// Mitsubishi GX Works2 project: 21   PLC: FX3G

// task Task_01 (event TRUE, interval 0, priority 31): POU_01

PROGRAM POU_01
VAR
  gas : INT;
  ton1 : TON;
END_VAR
IF M8002 THEN
	gas := 0;
END_IF;

	IF M0=TRUE THEN
	gas:=11;
END_IF;

IF M1=TRUE THEN
	gas:=21;
END_IF;

IF M2=TRUE THEN
	gas:=31;
END_IF;

CASE gas OF

	11:
	Y0:=TRUE;
	Y1:=FALSE;
	Y2:=FALSE;
	Y3:=FALSE;
	ton1(IN := NOT ton1.Q, PT := T#0.5s);
	IF ton1.Q THEN
		gas:=12;
	END_IF;
	
	12:
	Y0:=FALSE;
	Y1:=TRUE;
	Y2:=FALSE;
	Y3:=FALSE;
	ton1(IN := NOT ton1.Q, PT := T#0.5s);
	IF ton1.Q THEN
		gas:=13;
	END_IF;

 13:
	Y0:=FALSE;
	Y1:=FALSE;
	Y2:=TRUE;
	Y3:=FALSE;
	ton1(IN := NOT ton1.Q, PT := T#0.5s);
	IF ton1.Q THEN
		gas:=14;
	END_IF;
	
	14:
	Y0:=FALSE;
	Y1:=FALSE;
	Y2:=FALSE;
	Y3:=TRUE;
	ton1(IN := NOT ton1.Q, PT := T#0.5s);
	IF ton1.Q THEN
		gas:=11;
	END_IF;
	
	21:
	Y0:=TRUE;
	Y1:=FALSE;
	Y2:=FALSE;
	Y3:=FALSE;
	ton1(IN := NOT ton1.Q, PT := T#1s);
	IF ton1.Q THEN
		gas:=22;
	END_IF;
	
	22:
	Y0:=FALSE;
	Y1:=TRUE;
	Y2:=FALSE;
	Y3:=FALSE;
	ton1(IN := NOT ton1.Q, PT := T#1s);
	IF ton1.Q THEN
		gas:=23;
	END_IF;

 	23:
	Y0:=FALSE;
	Y1:=FALSE;
	Y2:=TRUE;
	Y3:=FALSE;
	ton1(IN := NOT ton1.Q, PT := T#1s);
	IF ton1.Q THEN
		gas:=24;
	END_IF;
	
	24:
	Y0:=FALSE;
	Y1:=FALSE;
	Y2:=FALSE;
	Y3:=TRUE;
	ton1(IN := NOT ton1.Q, PT := T#1s);
	IF ton1.Q THEN
		gas:=21;
	END_IF;
	
	31:
	Y0:=TRUE;
	Y1:=FALSE;
	Y2:=FALSE;
	Y3:=FALSE;
	ton1(IN := NOT ton1.Q, PT := T#1.5s);
	IF ton1.Q THEN
		gas:=32;
	END_IF;
	
	32:
	Y0:=FALSE;
	Y1:=TRUE;
	Y2:=FALSE;
	Y3:=FALSE;
	ton1(IN := NOT ton1.Q, PT := T#1.5s);
	IF ton1.Q THEN
		gas:=33;
	END_IF;

 	33:
	Y0:=FALSE;
	Y1:=FALSE;
	Y2:=TRUE;
	Y3:=FALSE;
	ton1(IN := NOT ton1.Q, PT := T#1.5s);
	IF ton1.Q THEN
		gas:=34;
	END_IF;
	
	34:
	Y0:=FALSE;
	Y1:=FALSE;
	Y2:=FALSE;
	Y3:=TRUE;
	ton1(IN := NOT ton1.Q, PT := T#1.5s);
	IF ton1.Q THEN
		gas:=31;
	END_IF;
	
	END_CASE;
END_PROGRAM
